Fanuc KAREL source: kt00264.KL

PROGRAM KT00264
%NOLOCKGROUP
VAR
R1:REAL
H2 : ARRAY[2] OF SHORT
OUT:BOOLEAN
BEGIN
R1=2.0
H2[1]=3
OUT=(R1=(H2[1]))
END KT00264
